FUNCTION_BLOCK FB_Actuator IMPLEMENTS ITF_Actuator
VAR
	AdvanceBit		: BOOL := FALSE;
	RetractBit		: BOOL := FALSE;
	
	AdvanceTimer	: TON;
	RetractTimer	: TON;
	
	{ attribute 'TcHmiSymbol.AddSymbol' }
	OperatorControl	: BOOL := FALSE; //HMI Operator Control (Actuator state reverts to original state when out of Op control)
	OpControlFTRIG	: F_TRIG;
	
	{ attribute 'TcHmiSymbol.AddSymbol' }
	OperatorValue	: E_ActuatorState; //HMI Operator Value
	HeldValue		: E_ActuatorState;
	
	HardwareOverride	: BOOL; //For engineering actuator overriding
	OverrideValue		: E_ActuatorState; //Override Value
END_VAR

VAR_INPUT
	AdvancedIN		: FB_DigitalInput;
	RetractedIN		: FB_DigitalInput;
	AdvanceOUT		: FB_DigitalOutput;
	RetractOUT		: FB_DigitalOutput;
END_VAR

AdvanceOUT();
RetractOUT();

AdvancedIN();
RetractedIN();

AdvanceTimer(IN := AdvanceBit, PT := T#0.06S);
AdvanceOUT.SetOutput(AdvanceTimer.Q);

RetractTimer(IN := RetractBit, PT := T#0.06S);
RetractOUT.SetOutput(RetractTimer.Q);

//Retain value prior to going into operator control
OpControlFTRIG(CLK := OperatorControl);
IF OpControlFTRIG.Q THEN
	IF HeldValue = E_ActuatorState.Advance THEN
		Advance();
	ELSIF HeldValue = E_ActuatorState.Retract THEN
		Retract();
	END_IF
END_IF

IF NOT OperatorControl AND NOT HardwareOverride AND AdvancedIN.P_Value THEN
	OperatorValue 	:= E_ActuatorState.Advance;
	OverrideValue	:= E_ActuatorState.Advance;
	HeldValue 		:= E_ActuatorState.Advance;
ELSIF NOT OperatorControl AND NOT HardwareOverride AND RetractedIN.P_Value THEN
	OperatorValue 	:= E_ActuatorState.Retract;
	OverrideValue	:= E_ActuatorState.Retract;
	HeldValue 		:= E_ActuatorState.Retract;
END_IF

IF OperatorControl THEN
	IF OperatorValue = E_ActuatorState.Advance THEN
		Advance();
	ELSIF OperatorValue = E_ActuatorState.Retract THEN
		Retract();
	END_IF
END_IF

IF HardwareOverride THEN
	IF OverrideValue = E_ActuatorState.Advance THEN
		Advance();
	ELSIF OverrideValue = E_ActuatorState.Retract THEN
		Retract();
	END_IF
END_IF

METHOD Advance
RetractOUT.SetOutput(FALSE);
RetractBit := FALSE;
AdvanceBit := TRUE;
END_METHOD

PROPERTY P_Advanced : BOOL
GET
P_Advanced := AdvancedIN.P_Value;
END_GET
END_PROPERTY

PROPERTY P_OperatorControl : BOOL
GET
P_OperatorControl := OperatorControl;
END_GET
SET
OperatorControl := P_OperatorControl;
END_SET
END_PROPERTY

PROPERTY P_OperatorValue : E_ActuatorState
GET
P_OperatorValue := OperatorValue;
END_GET
SET
OperatorValue := P_OperatorValue;
END_SET
END_PROPERTY

PROPERTY P_Retracted : BOOL
GET
P_Retracted := RetractedIN.P_Value;
END_GET
END_PROPERTY

METHOD Retract
AdvanceOUT.SetOutput(FALSE);
RetractBit := TRUE;
AdvanceBit := FALSE;
END_METHOD

END_FUNCTION_BLOCK

(* stored: Version 1.1.0.1
   POU FB_Actuator: Id {801d48b9-2a03-40e7-ad0e-7a6554a9514a}, SpecialFunc None
   Folder Methods: Id {e1218f82-608a-4612-b7fc-8bee389e1376}
   Folder Properties: Id {45f78a4f-dbfe-4094-b321-f7434392df06}
   Method Advance: Id {e32a0885-2c88-4733-b66e-9be8b3841b33}
   Property P_Advanced: Id {28164b35-a2e9-428c-a89a-c4d9c7d896ed}
   Get Get: Id {6930b750-5574-4f1d-81da-db6e02241df9}
   Property P_OperatorControl: Id {bca32f3c-f1c5-4276-b40b-068851080a38}
   Get Get: Id {dbe7d2be-9f35-4f7e-bf3a-add9325190d1}
   Set Set: Id {f69bb334-d219-474e-91ad-1dc5b4050baf}
   Property P_OperatorValue: Id {c58f1bf1-35b1-445e-8311-b593a5a0b576}
   Get Get: Id {795c3b5d-0137-4afd-895e-3da17e165b0c}
   Set Set: Id {39374a3e-ce01-4171-90bb-a2c2aab1ded2}
   Property P_Retracted: Id {6f8b76f0-7809-4e03-bb50-a652494c777d}
   Get Get: Id {b3c98f22-73e2-4670-a813-a8981ba1aa4b}
   Method Retract: Id {ab3b65ce-ede5-4f7b-87c5-83a5a71a87fa} *)
